INTERFACE ITcMessage_Ext

METHOD Send : BOOL
VAR_INPUT
	eventType : Tc3_EventLogger.TcEventEntry;
	args : STRING(255);
END_VAR
END_METHOD

END_INTERFACE

(* stored: Version 1.1.0.1
   Itf ITcMessage_Ext: Id {2099f939-9ec3-4558-8ed7-fb5fbee10ec9}
   Method Send: Id {98f2b7ce-6e57-4fac-ac6c-a2745891cfea} *)
